Fanuc KAREL source: NC0073.KL

-- PROVISIONAL review KL for V770-1; original PC SHA256 f970b011553cad6f6cd56b2b257962deb463e3bd78e2a16155022fbe553c0953
-- Incomplete behavior may be omitted. Consult companion uncertainty JSON. Do not deploy.
PROGRAM NC0073
%NOLOCKGROUP
-- UNRESOLVED_LOCAL_POOL 1 cells at code offset 3; source declarations unknown
-- DIRECT_LOCAL_WORD_ACCESS alone does not prove INTEGER, REAL, or BOOLEAN
BEGIN
  -- UNRESOLVED_PC offsets 0-8; opcodes 2B,2C,7B
  -- UNRESOLVED_PC offsets 13-20; opcodes 9D,23
  -- UNRESOLVED_PC offsets 25-42; opcodes 21,2E,59,79
  -- UNRESOLVED_PC offsets 47-64; opcodes 21,2E,59,79
  -- UNRESOLVED_PC offsets 69-83; opcodes 21,9D,52,23
  -- UNRESOLVED_PC offsets 88-93; opcodes 7A
  -- UNRESOLVED_PC offsets 98-103; opcodes 7A
  -- UNRESOLVED_PC offsets 108-112; opcodes 7F
  -- UNRESOLVED_PC offsets 117-121; opcodes 27,AA
  -- UNRESOLVED_PC offsets 126-130; opcodes 7F
END NC0073
